ABB RAPID module: Module1.mod

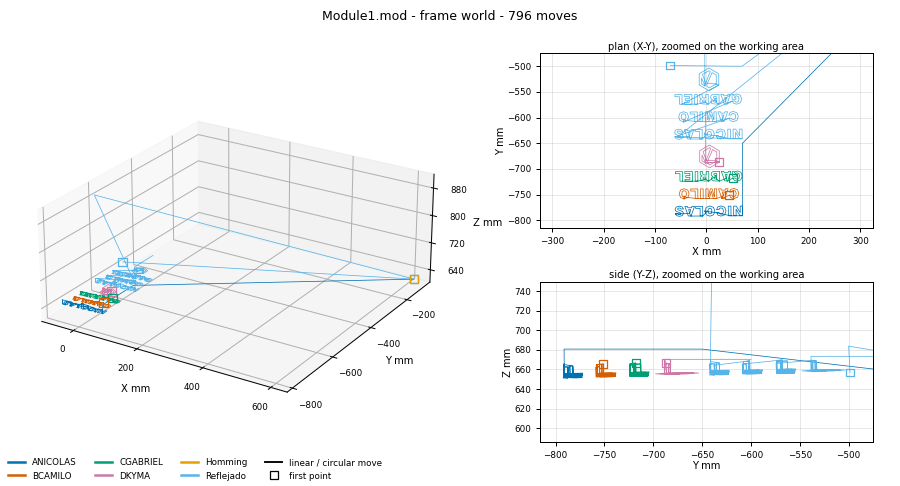
[picture p0: tool path of Module1.mod in frame world, 796 of 800 moves have a stored position in this frame; points joined in program order, loops and branches not executed]
MODULE Module1
    !CONST robtarget Target_10:=[[138.975,143.37,-10],[0.119542298,0.027125582,0.159127158,0.979618492],[-1,-1,1,0],[9E+09,9E+09,9E+09,9E+09,9E+09,9E+09]];
    CONST robtarget Target_10:=[[139.514118203,143.062380794,-24.987379073],[0.119542298,0.027125582,0.159127158,0.979618492],[-1,-1,1,0],[9E+09,9E+09,9E+09,9E+09,9E+09,9E+09]];
    CONST robtarget Target_20:=[[138.975,143.37,0],[0.119542298,0.027125582,0.159127158,0.979618492],[-1,-1,1,0],[9E+09,9E+09,9E+09,9E+09,9E+09,9E+09]];
    CONST robtarget Target_30:=[[133.906,143.37,0],[0.119542298,0.027125582,0.159127158,0.979618492],[-1,-1,1,0],[9E+09,9E+09,9E+09,9E+09,9E+09,9E+09]];
    CONST robtarget Target_40:=[[126.245,130.656,0],[0.119542298,0.027125582,0.159127158,0.979618492],[-1,-1,1,0],[9E+09,9E+09,9E+09,9E+09,9E+09,9E+09]];
    CONST robtarget Target_50:=[[126.245,143.37,0],[0.119542298,0.027125582,0.159127158,0.979618492],[-1,-1,1,0],[9E+09,9E+09,9E+09,9E+09,9E+09,9E+09]];
    CONST robtarget Target_60:=[[121.518,143.37,0],[0.119542298,0.027125582,0.159127158,0.979618492],[-1,-1,1,0],[9E+09,9E+09,9E+09,9E+09,9E+09,9E+09]];
    CONST robtarget Target_70:=[[121.518,124.69,0],[0.119542298,0.027125582,0.159127158,0.979618492],[-1,-1,1,0],[9E+09,9E+09,9E+09,9E+09,9E+09,9E+09]];
    CONST robtarget Target_80:=[[126.603,124.69,0],[0.119542298,0.027125582,0.159127158,0.979618492],[-1,-1,1,0],[9E+09,9E+09,9E+09,9E+09,9E+09,9E+09]];
    CONST robtarget Target_90:=[[134.248,137.371,0],[0.119542298,0.027125582,0.159127158,0.979618492],[-1,-1,1,0],[9E+09,9E+09,9E+09,9E+09,9E+09,9E+09]];
    CONST robtarget Target_100:=[[134.248,124.69,0],[0.119542298,0.027125582,0.159127158,0.979618492],[-1,-1,1,0],[9E+09,9E+09,9E+09,9E+09,9E+09,9E+09]];
    CONST robtarget Target_110:=[[138.975,124.69,0],[0.119542298,0.027125582,0.159127158,0.979618492],[-1,-1,1,0],[9E+09,9E+09,9E+09,9E+09,9E+09,9E+09]];
    CONST robtarget Target_120:=[[138.975,143.37,0],[0.119542298,0.027125582,0.159127158,0.979618492],[-1,-1,1,0],[9E+09,9E+09,9E+09,9E+09,9E+09,9E+09]];
    CONST robtarget Target_130:=[[138.975,143.37,-10],[0.119542298,0.027125582,0.159127158,0.979618492],[-1,-1,1,0],[9E+09,9E+09,9E+09,9E+09,9E+09,9E+09]];
    CONST robtarget Target_140:=[[116.236,143.37,-10],[0.119542298,0.027125582,0.159127158,0.979618492],[-1,-1,1,0],[9E+09,9E+09,9E+09,9E+09,9E+09,9E+09]];
    CONST robtarget Target_150:=[[116.236,143.37,0],[0.119542298,0.027125582,0.159127158,0.979618492],[-1,-1,1,0],[9E+09,9E+09,9E+09,9E+09,9E+09,9E+09]];
    CONST robtarget Target_160:=[[111.069,143.37,0],[0.119542298,0.027125582,0.159127158,0.979618492],[-1,-1,1,0],[9E+09,9E+09,9E+09,9E+09,9E+09,9E+09]];
    CONST robtarget Target_170:=[[111.069,124.69,0],[0.119542298,0.027125582,0.159127158,0.979618492],[-1,-1,1,0],[9E+09,9E+09,9E+09,9E+09,9E+09,9E+09]];
    CONST robtarget Target_180:=[[116.236,124.69,0],[0.119542298,0.027125582,0.159127158,0.979618492],[-1,-1,1,0],[9E+09,9E+09,9E+09,9E+09,9E+09,9E+09]];
    CONST robtarget Target_190:=[[116.236,143.37,0],[0.119542298,0.027125582,0.159127158,0.979618492],[-1,-1,1,0],[9E+09,9E+09,9E+09,9E+09,9E+09,9E+09]];
    CONST robtarget Target_200:=[[116.236,143.37,-10],[0.119542298,0.027125582,0.159127158,0.979618492],[-1,-1,1,0],[9E+09,9E+09,9E+09,9E+09,9E+09,9E+09]];
    CONST robtarget Target_210:=[[88.445,137.143,-10],[0.119542298,0.027125582,0.159127158,0.979618492],[-1,-1,1,0],[9E+09,9E+09,9E+09,9E+09,9E+09,9E+09]];
    CONST robtarget Target_220:=[[88.445,137.143,0],[0.119542298,0.027125582,0.159127158,0.979618492],[-1,-1,1,0],[9E+09,9E+09,9E+09,9E+09,9E+09,9E+09]];
    CONST robtarget Target_230:=[[90.98,142.156,0],[0.119542298,0.027125582,0.159127158,0.979618492],[-1,-1,1,0],[9E+09,9E+09,9E+09,9E+09,9E+09,9E+09]];
    CONST robtarget Target_240:=[[96.97,143.973,0],[0.119542298,0.027125582,0.159127158,0.979618492],[-1,-1,1,0],[9E+09,9E+09,9E+09,9E+09,9E+09,9E+09]];
    CONST robtarget Target_250:=[[104.06,141.341,0],[0.119542298,0.027125582,0.159127158,0.979618492],[-1,-1,1,0],[9E+09,9E+09,9E+09,9E+09,9E+09,9E+09]];
    CONST robtarget Target_260:=[[106.62,134.046,0],[0.119542298,0.027125582,0.159127158,0.979618492],[-1,-1,1,0],[9E+09,9E+09,9E+09,9E+09,9E+09,9E+09]];
    CONST robtarget Target_270:=[[104.077,126.752,0],[0.119542298,0.027125582,0.159127158,0.979618492],[-1,-1,1,0],[9E+09,9E+09,9E+09,9E+09,9E+09,9E+09]];
    CONST robtarget Target_280:=[[96.954,124.136,0],[0.119542298,0.027125582,0.159127158,0.979618492],[-1,-1,1,0],[9E+09,9E+09,9E+09,9E+09,9E+09,9E+09]];
    CONST robtarget Target_290:=[[90.866,125.978,0],[0.119542298,0.027125582,0.159127158,0.979618492],[-1,-1,1,0],[9E+09,9E+09,9E+09,9E+09,9E+09,9E+09]];
    CONST robtarget Target_300:=[[88.201,131.178,0],[0.119542298,0.027125582,0.159127158,0.979618492],[-1,-1,1,0],[9E+09,9E+09,9E+09,9E+09,9E+09,9E+09]];
    CONST robtarget Target_310:=[[90.556,131.178,0],[0.119542298,0.027125582,0.159127158,0.979618492],[-1,-1,1,0],[9E+09,9E+09,9E+09,9E+09,9E+09,9E+09]];
    CONST robtarget Target_320:=[[92.911,131.178,0],[0.119542298,0.027125582,0.159127158,0.979618492],[-1,-1,1,0],[9E+09,9E+09,9E+09,9E+09,9E+09,9E+09]];
    CONST robtarget Target_330:=[[94.207,128.781,0],[0.119542298,0.027125582,0.159127158,0.979618492],[-1,-1,1,0],[9E+09,9E+09,9E+09,9E+09,9E+09,9E+09]];
    CONST robtarget Target_340:=[[96.937,127.885,0],[0.119542298,0.027125582,0.159127158,0.979618492],[-1,-1,1,0],[9E+09,9E+09,9E+09,9E+09,9E+09,9E+09]];
    CONST robtarget Target_350:=[[100.385,129.458,0],[0.119542298,0.027125582,0.159127158,0.979618492],[-1,-1,1,0],[9E+09,9E+09,9E+09,9E+09,9E+09,9E+09]];
    CONST robtarget Target_360:=[[101.583,134.03,0],[0.119542298,0.027125582,0.159127158,0.979618492],[-1,-1,1,0],[9E+09,9E+09,9E+09,9E+09,9E+09,9E+09]];
    CONST robtarget Target_370:=[[100.426,138.635,0],[0.119542298,0.027125582,0.159127158,0.979618492],[-1,-1,1,0],[9E+09,9E+09,9E+09,9E+09,9E+09,9E+09]];
    CONST robtarget Target_380:=[[96.937,140.175,0],[0.119542298,0.027125582,0.159127158,0.979618492],[-1,-1,1,0],[9E+09,9E+09,9E+09,9E+09,9E+09,9E+09]];
    CONST robtarget Target_390:=[[94.329,139.376,0],[0.119542298,0.027125582,0.159127158,0.979618492],[-1,-1,1,0],[9E+09,9E+09,9E+09,9E+09,9E+09,9E+09]];
    CONST robtarget Target_400:=[[93.058,137.143,0],[0.119542298,0.027125582,0.159127158,0.979618492],[-1,-1,1,0],[9E+09,9E+09,9E+09,9E+09,9E+09,9E+09]];
    CONST robtarget Target_410:=[[90.752,137.143,0],[0.119542298,0.027125582,0.159127158,0.979618492],[-1,-1,1,0],[9E+09,9E+09,9E+09,9E+09,9E+09,9E+09]];
    CONST robtarget Target_420:=[[88.445,137.143,0],[0.119542298,0.027125582,0.159127158,0.979618492],[-1,-1,1,0],[9E+09,9E+09,9E+09,9E+09,9E+09,9E+09]];
    CONST robtarget Target_430:=[[88.445,137.143,-10],[0.119542298,0.027125582,0.159127158,0.979618492],[-1,-1,1,0],[9E+09,9E+09,9E+09,9E+09,9E+09,9E+09]];
    CONST robtarget Target_440:=[[65.511,134.046,-10],[0.119542298,0.027125582,0.159127158,0.979618492],[-1,-1,1,0],[9E+09,9E+09,9E+09,9E+09,9E+09,9E+09]];
    CONST robtarget Target_450:=[[65.511,134.046,0],[0.119542298,0.027125582,0.159127158,0.979618492],[-1,-1,1,0],[9E+09,9E+09,9E+09,9E+09,9E+09,9E+09]];
    CONST robtarget Target_460:=[[68.127,141.3,0],[0.119542298,0.027125582,0.159127158,0.979618492],[-1,-1,1,0],[9E+09,9E+09,9E+09,9E+09,9E+09,9E+09]];
    CONST robtarget Target_470:=[[75.21,143.973,0],[0.119542298,0.027125582,0.159127158,0.979618492],[-1,-1,1,0],[9E+09,9E+09,9E+09,9E+09,9E+09,9E+09]];
    CONST robtarget Target_480:=[[82.3,141.3,0],[0.119542298,0.027125582,0.159127158,0.979618492],[-1,-1,1,0],[9E+09,9E+09,9E+09,9E+09,9E+09,9E+09]];
    CONST robtarget Target_490:=[[84.908,134.046,0],[0.119542298,0.027125582,0.159127158,0.979618492],[-1,-1,1,0],[9E+09,9E+09,9E+09,9E+09,9E+09,9E+09]];
    CONST robtarget Target_500:=[[82.3,126.809,0],[0.119542298,0.027125582,0.159127158,0.979618492],[-1,-1,1,0],[9E+09,9E+09,9E+09,9E+09,9E+09,9E+09]];
    CONST robtarget Target_510:=[[75.21,124.136,0],[0.119542298,0.027125582,0.159127158,0.979618492],[-1,-1,1,0],[9E+09,9E+09,9E+09,9E+09,9E+09,9E+09]];
    CONST robtarget Target_520:=[[68.119,126.809,0],[0.119542298,0.027125582,0.159127158,0.979618492],[-1,-1,1,0],[9E+09,9E+09,9E+09,9E+09,9E+09,9E+09]];
    CONST robtarget Target_530:=[[65.511,134.046,0],[0.119542298,0.027125582,0.159127158,0.979618492],[-1,-1,1,0],[9E+09,9E+09,9E+09,9E+09,9E+09,9E+09]];
    CONST robtarget Target_540:=[[65.511,134.046,-10],[0.119542298,0.027125582,0.159127158,0.979618492],[-1,-1,1,0],[9E+09,9E+09,9E+09,9E+09,9E+09,9E+09]];
    CONST robtarget Target_550:=[[71.298,134.046,-10],[0.119542298,0.027125582,0.159127158,0.979618492],[-1,-1,1,0],[9E+09,9E+09,9E+09,9E+09,9E+09,9E+09]];
    CONST robtarget Target_560:=[[71.298,134.046,0],[0.119542298,0.027125582,0.159127158,0.979618492],[-1,-1,1,0],[9E+09,9E+09,9E+09,9E+09,9E+09,9E+09]];
    CONST robtarget Target_570:=[[72.235,129.865,0],[0.119542298,0.027125582,0.159127158,0.979618492],[-1,-1,1,0],[9E+09,9E+09,9E+09,9E+09,9E+09,9E+09]];
    CONST robtarget Target_580:=[[75.193,128.537,0],[0.119542298,0.027125582,0.159127158,0.979618492],[-1,-1,1,0],[9E+09,9E+09,9E+09,9E+09,9E+09,9E+09]];
    CONST robtarget Target_590:=[[78.176,129.865,0],[0.119542298,0.027125582,0.159127158,0.979618492],[-1,-1,1,0],[9E+09,9E+09,9E+09,9E+09,9E+09,9E+09]];
    CONST robtarget Target_600:=[[79.122,134.046,0],[0.119542298,0.027125582,0.159127158,0.979618492],[-1,-1,1,0],[9E+09,9E+09,9E+09,9E+09,9E+09,9E+09]];
    CONST robtarget Target_610:=[[78.176,138.227,0],[0.119542298,0.027125582,0.159127158,0.979618492],[-1,-1,1,0],[9E+09,9E+09,9E+09,9E+09,9E+09,9E+09]];
    CONST robtarget Target_620:=[[75.193,139.556,0],[0.119542298,0.027125582,0.159127158,0.979618492],[-1,-1,1,0],[9E+09,9E+09,9E+09,9E+09,9E+09,9E+09]];
    CONST robtarget Target_630:=[[72.235,138.227,0],[0.119542298,0.027125582,0.159127158,0.979618492],[-1,-1,1,0],[9E+09,9E+09,9E+09,9E+09,9E+09,9E+09]];
    CONST robtarget Target_640:=[[71.298,134.046,0],[0.119542298,0.027125582,0.159127158,0.979618492],[-1,-1,1,0],[9E+09,9E+09,9E+09,9E+09,9E+09,9E+09]];
    CONST robtarget Target_650:=[[71.298,134.046,-10],[0.119542298,0.027125582,0.159127158,0.979618492],[-1,-1,1,0],[9E+09,9E+09,9E+09,9E+09,9E+09,9E+09]];
    CONST robtarget Target_660:=[[61.192,143.37,-10],[0.119542298,0.027125582,0.159127158,0.979618492],[-1,-1,1,0],[9E+09,9E+09,9E+09,9E+09,9E+09,9E+09]];
    CONST robtarget Target_670:=[[61.192,143.37,0],[0.119542298,0.027125582,0.159127158,0.979618492],[-1,-1,1,0],[9E+09,9E+09,9E+09,9E+09,9E+09,9E+09]];
    CONST robtarget Target_680:=[[56.139,143.37,0],[0.119542298,0.027125582,0.159127158,0.979618492],[-1,-1,1,0],[9E+09,9E+09,9E+09,9E+09,9E+09,9E+09]];
    CONST robtarget Target_690:=[[56.139,128.7,0],[0.119542298,0.027125582,0.159127158,0.979618492],[-1,-1,1,0],[9E+09,9E+09,9E+09,9E+09,9E+09,9E+09]];
    CONST robtarget Target_700:=[[47.402,128.7,0],[0.119542298,0.027125582,0.159127158,0.979618492],[-1,-1,1,0],[9E+09,9E+09,9E+09,9E+09,9E+09,9E+09]];
    CONST robtarget Target_710:=[[47.402,124.69,0],[0.119542298,0.027125582,0.159127158,0.979618492],[-1,-1,1,0],[9E+09,9E+09,9E+09,9E+09,9E+09,9E+09]];
    CONST robtarget Target_720:=[[61.192,124.69,0],[0.119542298,0.027125582,0.159127158,0.979618492],[-1,-1,1,0],[9E+09,9E+09,9E+09,9E+09,9E+09,9E+09]];
    CONST robtarget Target_730:=[[61.192,143.37,0],[0.119542298,0.027125582,0.159127158,0.979618492],[-1,-1,1,0],[9E+09,9E+09,9E+09,9E+09,9E+09,9E+09]];
    CONST robtarget Target_740:=[[61.192,143.37,-10],[0.119542298,0.027125582,0.159127158,0.979618492],[-1,-1,1,0],[9E+09,9E+09,9E+09,9E+09,9E+09,9E+09]];
    CONST robtarget Target_750:=[[38.567,143.37,-10],[0.119542298,0.027125582,0.159127158,0.979618492],[-1,-1,1,0],[9E+09,9E+09,9E+09,9E+09,9E+09,9E+09]];
    CONST robtarget Target_760:=[[38.567,143.37,0],[0.119542298,0.027125582,0.159127158,0.979618492],[-1,-1,1,0],[9E+09,9E+09,9E+09,9E+09,9E+09,9E+09]];
    CONST robtarget Target_770:=[[33.025,143.37,0],[0.119542298,0.027125582,0.159127158,0.979618492],[-1,-1,1,0],[9E+09,9E+09,9E+09,9E+09,9E+09,9E+09]];
    CONST robtarget Target_780:=[[26.424,124.69,0],[0.119542298,0.027125582,0.159127158,0.979618492],[-1,-1,1,0],[9E+09,9E+09,9E+09,9E+09,9E+09,9E+09]];
    CONST robtarget Target_790:=[[31.412,124.69,0],[0.119542298,0.027125582,0.159127158,0.979618492],[-1,-1,1,0],[9E+09,9E+09,9E+09,9E+09,9E+09,9E+09]];
    CONST robtarget Target_800:=[[32.178,127.331,0],[0.119542298,0.027125582,0.159127158,0.979618492],[-1,-1,1,0],[9E+09,9E+09,9E+09,9E+09,9E+09,9E+09]];
    CONST robtarget Target_810:=[[39.464,127.331,0],[0.119542298,0.027125582,0.159127158,0.979618492],[-1,-1,1,0],[9E+09,9E+09,9E+09,9E+09,9E+09,9E+09]];
    CONST robtarget Target_820:=[[40.181,124.69,0],[0.119542298,0.027125582,0.159127158,0.979618492],[-1,-1,1,0],[9E+09,9E+09,9E+09,9E+09,9E+09,9E+09]];
    CONST robtarget Target_830:=[[45.169,124.69,0],[0.119542298,0.027125582,0.159127158,0.979618492],[-1,-1,1,0],[9E+09,9E+09,9E+09,9E+09,9E+09,9E+09]];
    CONST robtarget Target_840:=[[38.567,143.37,0],[0.119542298,0.027125582,0.159127158,0.979618492],[-1,-1,1,0],[9E+09,9E+09,9E+09,9E+09,9E+09,9E+09]];
    CONST robtarget Target_850:=[[38.567,143.37,-10],[0.119542298,0.027125582,0.159127158,0.979618492],[-1,-1,1,0],[9E+09,9E+09,9E+09,9E+09,9E+09,9E+09]];
    CONST robtarget Target_860:=[[35.796,138.464,-10],[0.119542298,0.027125582,0.159127158,0.979618492],[-1,-1,1,0],[9E+09,9E+09,9E+09,9E+09,9E+09,9E+09]];
    CONST robtarget Target_870:=[[35.796,138.464,0],[0.119542298,0.027125582,0.159127158,0.979618492],[-1,-1,1,0],[9E+09,9E+09,9E+09,9E+09,9E+09,9E+09]];
    CONST robtarget Target_880:=[[37.834,130.884,0],[0.119542298,0.027125582,0.159127158,0.979618492],[-1,-1,1,0],[9E+09,9E+09,9E+09,9E+09,9E+09,9E+09]];
    CONST robtarget Target_890:=[[33.791,130.884,0],[0.119542298,0.027125582,0.159127158,0.979618492],[-1,-1,1,0],[9E+09,9E+09,9E+09,9E+09,9E+09,9E+09]];
    CONST robtarget Target_900:=[[35.796,138.464,0],[0.119542298,0.027125582,0.159127158,0.979618492],[-1,-1,1,0],[9E+09,9E+09,9E+09,9E+09,9E+09,9E+09]];
    CONST robtarget Target_910:=[[35.796,138.464,-10],[0.119542298,0.027125582,0.159127158,0.979618492],[-1,-1,1,0],[9E+09,9E+09,9E+09,9E+09,9E+09,9E+09]];
    CONST robtarget Target_920:=[[8.038,138.936,-10],[0.119542298,0.027125582,0.159127158,0.979618492],[-1,-1,1,0],[9E+09,9E+09,9E+09,9E+09,9E+09,9E+09]];
    CONST robtarget Target_930:=[[8.038,138.936,0],[0.119542298,0.027125582,0.159127158,0.979618492],[-1,-1,1,0],[9E+09,9E+09,9E+09,9E+09,9E+09,9E+09]];
    CONST robtarget Target_940:=[[10.58,142.702,0],[0.119542298,0.027125582,0.159127158,0.979618492],[-1,-1,1,0],[9E+09,9E+09,9E+09,9E+09,9E+09,9E+09]];
    CONST robtarget Target_950:=[[16.057,143.973,0],[0.119542298,0.027125582,0.159127158,0.979618492],[-1,-1,1,0],[9E+09,9E+09,9E+09,9E+09,9E+09,9E+09]];
    CONST robtarget Target_960:=[[21.558,142.416,0],[0.119542298,0.027125582,0.159127158,0.979618492],[-1,-1,1,0],[9E+09,9E+09,9E+09,9E+09,9E+09,9E+09]];
    CONST robtarget Target_970:=[[23.588,138.219,0],[0.119542298,0.027125582,0.159127158,0.979618492],[-1,-1,1,0],[9E+09,9E+09,9E+09,9E+09,9E+09,9E+09]];
    CONST robtarget Target_980:=[[22.267,134.812,0],[0.119542298,0.027125582,0.159127158,0.979618492],[-1,-1,1,0],[9E+09,9E+09,9E+09,9E+09,9E+09,9E+09]];
    CONST robtarget Target_990:=[[16.611,132.4,0],[0.119542298,0.027125582,0.159127158,0.979618492],[-1,-1,1,0],[9E+09,9E+09,9E+09,9E+09,9E+09,9E+09]];
    CONST robtarget Target_1000:=[[13.16,131.12,0],[0.119542298,0.027125582,0.159127158,0.979618492],[-1,-1,1,0],[9E+09,9E+09,9E+09,9E+09,9E+09,9E+09]];
    CONST robtarget Target_1010:=[[12.324,129.743,0],[0.119542298,0.027125582,0.159127158,0.979618492],[-1,-1,1,0],[9E+09,9E+09,9E+09,9E+09,9E+09,9E+09]];
    CONST robtarget Target_1020:=[[13.172,128.17,0],[0.119542298,0.027125582,0.159127158,0.979618492],[-1,-1,1,0],[9E+09,9E+09,9E+09,9E+09,9E+09,9E+09]];
    CONST robtarget Target_1030:=[[15.633,127.624,0],[0.119542298,0.027125582,0.159127158,0.979618492],[-1,-1,1,0],[9E+09,9E+09,9E+09,9E+09,9E+09,9E+09]];
    CONST robtarget Target_1040:=[[17.858,128.129,0],[0.119542298,0.027125582,0.159127158,0.979618492],[-1,-1,1,0],[9E+09,9E+09,9E+09,9E+09,9E+09,9E+09]];
    CONST robtarget Target_1050:=[[18.926,129.629,0],[0.119542298,0.027125582,0.159127158,0.979618492],[-1,-1,1,0],[9E+09,9E+09,9E+09,9E+09,9E+09,9E+09]];
    CONST robtarget Target_1060:=[[23.783,129.629,0],[0.119542298,0.027125582,0.159127158,0.979618492],[-1,-1,1,0],[9E+09,9E+09,9E+09,9E+09,9E+09,9E+09]];
    CONST robtarget Target_1070:=[[21.192,125.587,0],[0.119542298,0.027125582,0.159127158,0.979618492],[-1,-1,1,0],[9E+09,9E+09,9E+09,9E+09,9E+09,9E+09]];
    CONST robtarget Target_1080:=[[15.715,124.169,0],[0.119542298,0.027125582,0.159127158,0.979618492],[-1,-1,1,0],[9E+09,9E+09,9E+09,9E+09,9E+09,9E+09]];
    CONST robtarget Target_1090:=[[9.554,125.741,0],[0.119542298,0.027125582,0.159127158,0.979618492],[-1,-1,1,0],[9E+09,9E+09,9E+09,9E+09,9E+09,9E+09]];
    CONST robtarget Target_1100:=[[7.451,130.379,0],[0.119542298,0.027125582,0.159127158,0.979618492],[-1,-1,1,0],[9E+09,9E+09,9E+09,9E+09,9E+09,9E+09]];
    CONST robtarget Target_1110:=[[8.885,133.875,0],[0.119542298,0.027125582,0.159127158,0.979618492],[-1,-1,1,0],[9E+09,9E+09,9E+09,9E+09,9E+09,9E+09]];
    CONST robtarget Target_1120:=[[15.03,136.328,0],[0.119542298,0.027125582,0.159127158,0.979618492],[-1,-1,1,0],[9E+09,9E+09,9E+09,9E+09,9E+09,9E+09]];
    CONST robtarget Target_1130:=[[17.85,137.412,0],[0.119542298,0.027125582,0.159127158,0.979618492],[-1,-1,1,0],[9E+09,9E+09,9E+09,9E+09,9E+09,9E+09]];
    CONST robtarget Target_1140:=[[18.698,138.773,0],[0.119542298,0.027125582,0.159127158,0.979618492],[-1,-1,1,0],[9E+09,9E+09,9E+09,9E+09,9E+09,9E+09]];
    CONST robtarget Target_1150:=[[17.972,140.208,0],[0.119542298,0.027125582,0.159127158,0.979618492],[-1,-1,1,0],[9E+09,9E+09,9E+09,9E+09,9E+09,9E+09]];
    CONST robtarget Target_1160:=[[15.976,140.729,0],[0.119542298,0.027125582,0.159127158,0.979618492],[-1,-1,1,0],[9E+09,9E+09,9E+09,9E+09,9E+09,9E+09]];
    CONST robtarget Target_1170:=[[13.889,140.265,0],[0.119542298,0.027125582,0.159127158,0.979618492],[-1,-1,1,0],[9E+09,9E+09,9E+09,9E+09,9E+09,9E+09]];
    CONST robtarget Target_1180:=[[12.879,138.936,0],[0.119542298,0.027125582,0.159127158,0.979618492],[-1,-1,1,0],[9E+09,9E+09,9E+09,9E+09,9E+09,9E+09]];
    CONST robtarget Target_1190:=[[8.038,138.936,0],[0.119542298,0.027125582,0.159127158,0.979618492],[-1,-1,1,0],[9E+09,9E+09,9E+09,9E+09,9E+09,9E+09]];
    CONST robtarget Target_1200:=[[8.038,138.936,-10],[0.119542298,0.027125582,0.159127158,0.979618492],[-1,-1,1,0],[9E+09,9E+09,9E+09,9E+09,9E+09,9E+09]];
    CONST robtarget Target_1210:=[[113.571,103.208,-10],[0.119542298,0.027125582,0.159127158,0.979618492],[-1,-1,1,0],[9E+09,9E+09,9E+09,9E+09,9E+09,9E+09]];
    CONST robtarget Target_1220:=[[113.571,103.208,0],[0.119542298,0.027125582,0.159127158,0.979618492],[-1,-1,1,0],[9E+09,9E+09,9E+09,9E+09,9E+09,9E+09]];
    CONST robtarget Target_1230:=[[116.106,108.22,0],[0.119542298,0.027125582,0.159127158,0.979618492],[-1,-1,1,0],[9E+09,9E+09,9E+09,9E+09,9E+09,9E+09]];
    CONST robtarget Target_1240:=[[122.096,110.037,0],[0.119542298,0.027125582,0.159127158,0.979618492],[-1,-1,1,0],[9E+09,9E+09,9E+09,9E+09,9E+09,9E+09]];
    CONST robtarget Target_1250:=[[129.187,107.405,0],[0.119542298,0.027125582,0.159127158,0.979618492],[-1,-1,1,0],[9E+09,9E+09,9E+09,9E+09,9E+09,9E+09]];
    CONST robtarget Target_1260:=[[131.746,100.111,0],[0.119542298,0.027125582,0.159127158,0.979618492],[-1,-1,1,0],[9E+09,9E+09,9E+09,9E+09,9E+09,9E+09]];
    CONST robtarget Target_1270:=[[129.203,92.817,0],[0.119542298,0.027125582,0.159127158,0.979618492],[-1,-1,1,0],[9E+09,9E+09,9E+09,9E+09,9E+09,9E+09]];
    CONST robtarget Target_1280:=[[122.08,90.2,0],[0.119542298,0.027125582,0.159127158,0.979618492],[-1,-1,1,0],[9E+09,9E+09,9E+09,9E+09,9E+09,9E+09]];
    CONST robtarget Target_1290:=[[115.992,92.042,0],[0.119542298,0.027125582,0.159127158,0.979618492],[-1,-1,1,0],[9E+09,9E+09,9E+09,9E+09,9E+09,9E+09]];
    CONST robtarget Target_1300:=[[113.327,97.242,0],[0.119542298,0.027125582,0.159127158,0.979618492],[-1,-1,1,0],[9E+09,9E+09,9E+09,9E+09,9E+09,9E+09]];
    CONST robtarget Target_1310:=[[118.038,97.242,0],[0.119542298,0.027125582,0.159127158,0.979618492],[-1,-1,1,0],[9E+09,9E+09,9E+09,9E+09,9E+09,9E+09]];
    CONST robtarget Target_1320:=[[119.333,94.846,0],[0.119542298,0.027125582,0.159127158,0.979618492],[-1,-1,1,0],[9E+09,9E+09,9E+09,9E+09,9E+09,9E+09]];
    CONST robtarget Target_1330:=[[122.064,93.949,0],[0.119542298,0.027125582,0.159127158,0.979618492],[-1,-1,1,0],[9E+09,9E+09,9E+09,9E+09,9E+09,9E+09]];
    CONST robtarget Target_1340:=[[125.511,95.522,0],[0.119542298,0.027125582,0.159127158,0.979618492],[-1,-1,1,0],[9E+09,9E+09,9E+09,9E+09,9E+09,9E+09]];
    CONST robtarget Target_1350:=[[126.709,100.094,0],[0.119542298,0.027125582,0.159127158,0.979618492],[-1,-1,1,0],[9E+09,9E+09,9E+09,9E+09,9E+09,9E+09]];
    CONST robtarget Target_1360:=[[125.552,104.699,0],[0.119542298,0.027125582,0.159127158,0.979618492],[-1,-1,1,0],[9E+09,9E+09,9E+09,9E+09,9E+09,9E+09]];
    CONST robtarget Target_1370:=[[122.064,106.239,0],[0.119542298,0.027125582,0.159127158,0.979618492],[-1,-1,1,0],[9E+09,9E+09,9E+09,9E+09,9E+09,9E+09]];
    CONST robtarget Target_1380:=[[119.456,105.441,0],[0.119542298,0.027125582,0.159127158,0.979618492],[-1,-1,1,0],[9E+09,9E+09,9E+09,9E+09,9E+09,9E+09]];
    CONST robtarget Target_1390:=[[118.184,103.208,0],[0.119542298,0.027125582,0.159127158,0.979618492],[-1,-1,1,0],[9E+09,9E+09,9E+09,9E+09,9E+09,9E+09]];
    CONST robtarget Target_1400:=[[113.571,103.208,0],[0.119542298,0.027125582,0.159127158,0.979618492],[-1,-1,1,0],[9E+09,9E+09,9E+09,9E+09,9E+09,9E+09]];
    CONST robtarget Target_1410:=[[113.571,103.208,-10],[0.119542298,0.027125582,0.159127158,0.979618492],[-1,-1,1,0],[9E+09,9E+09,9E+09,9E+09,9E+09,9E+09]];
    CONST robtarget Target_1420:=[[98.771,109.434,-10],[0.119542298,0.027125582,0.159127158,0.979618492],[-1,-1,1,0],[9E+09,9E+09,9E+09,9E+09,9E+09,9E+09]];
    CONST robtarget Target_1430:=[[98.771,109.434,0],[0.119542298,0.027125582,0.159127158,0.979618492],[-1,-1,1,0],[9E+09,9E+09,9E+09,9E+09,9E+09,9E+09]];
    CONST robtarget Target_1440:=[[92.17,90.755,0],[0.119542298,0.027125582,0.159127158,0.979618492],[-1,-1,1,0],[9E+09,9E+09,9E+09,9E+09,9E+09,9E+09]];
    CONST robtarget Target_1450:=[[97.157,90.755,0],[0.119542298,0.027125582,0.159127158,0.979618492],[-1,-1,1,0],[9E+09,9E+09,9E+09,9E+09,9E+09,9E+09]];
    CONST robtarget Target_1460:=[[97.924,93.395,0],[0.119542298,0.027125582,0.159127158,0.979618492],[-1,-1,1,0],[9E+09,9E+09,9E+09,9E+09,9E+09,9E+09]];
    CONST robtarget Target_1470:=[[105.21,93.395,0],[0.119542298,0.027125582,0.159127158,0.979618492],[-1,-1,1,0],[9E+09,9E+09,9E+09,9E+09,9E+09,9E+09]];
    CONST robtarget Target_1480:=[[105.927,90.755,0],[0.119542298,0.027125582,0.159127158,0.979618492],[-1,-1,1,0],[9E+09,9E+09,9E+09,9E+09,9E+09,9E+09]];
    CONST robtarget Target_1490:=[[110.915,90.755,0],[0.119542298,0.027125582,0.159127158,0.979618492],[-1,-1,1,0],[9E+09,9E+09,9E+09,9E+09,9E+09,9E+09]];
    CONST robtarget Target_1500:=[[104.313,109.434,0],[0.119542298,0.027125582,0.159127158,0.979618492],[-1,-1,1,0],[9E+09,9E+09,9E+09,9E+09,9E+09,9E+09]];
    CONST robtarget Target_1510:=[[98.771,109.434,0],[0.119542298,0.027125582,0.159127158,0.979618492],[-1,-1,1,0],[9E+09,9E+09,9E+09,9E+09,9E+09,9E+09]];
    CONST robtarget Target_1520:=[[98.771,109.434,-10],[0.119542298,0.027125582,0.159127158,0.979618492],[-1,-1,1,0],[9E+09,9E+09,9E+09,9E+09,9E+09,9E+09]];
    CONST robtarget Target_1530:=[[101.542,104.528,-10],[0.119542298,0.027125582,0.159127158,0.979618492],[-1,-1,1,0],[9E+09,9E+09,9E+09,9E+09,9E+09,9E+09]];
    CONST robtarget Target_1540:=[[101.542,104.528,0],[0.119542298,0.027125582,0.159127158,0.979618492],[-1,-1,1,0],[9E+09,9E+09,9E+09,9E+09,9E+09,9E+09]];
    CONST robtarget Target_1550:=[[103.58,96.949,0],[0.119542298,0.027125582,0.159127158,0.979618492],[-1,-1,1,0],[9E+09,9E+09,9E+09,9E+09,9E+09,9E+09]];
    CONST robtarget Target_1560:=[[99.537,96.949,0],[0.119542298,0.027125582,0.159127158,0.979618492],[-1,-1,1,0],[9E+09,9E+09,9E+09,9E+09,9E+09,9E+09]];
    CONST robtarget Target_1570:=[[101.542,104.528,0],[0.119542298,0.027125582,0.159127158,0.979618492],[-1,-1,1,0],[9E+09,9E+09,9E+09,9E+09,9E+09,9E+09]];
    CONST robtarget Target_1580:=[[101.542,104.528,-10],[0.119542298,0.027125582,0.159127158,0.979618492],[-1,-1,1,0],[9E+09,9E+09,9E+09,9E+09,9E+09,9E+09]];
    CONST robtarget Target_1590:=[[88.747,109.434,-10],[0.119542298,0.027125582,0.159127158,0.979618492],[-1,-1,1,0],[9E+09,9E+09,9E+09,9E+09,9E+09,9E+09]];
    CONST robtarget Target_1600:=[[88.747,109.434,0],[0.119542298,0.027125582,0.159127158,0.979618492],[-1,-1,1,0],[9E+09,9E+09,9E+09,9E+09,9E+09,9E+09]];
    CONST robtarget Target_1610:=[[88.747,90.755,0],[0.119542298,0.027125582,0.159127158,0.979618492],[-1,-1,1,0],[9E+09,9E+09,9E+09,9E+09,9E+09,9E+09]];
    CONST robtarget Target_1620:=[[84.297,90.755,0],[0.119542298,0.027125582,0.159127158,0.979618492],[-1,-1,1,0],[9E+09,9E+09,9E+09,9E+09,9E+09,9E+09]];
    CONST robtarget Target_1630:=[[84.297,105.848,0],[0.119542298,0.027125582,0.159127158,0.979618492],[-1,-1,1,0],[9E+09,9E+09,9E+09,9E+09,9E+09,9E+09]];
    CONST robtarget Target_1640:=[[83.743,105.848,0],[0.119542298,0.027125582,0.159127158,0.979618492],[-1,-1,1,0],[9E+09,9E+09,9E+09,9E+09,9E+09,9E+09]];
    CONST robtarget Target_1650:=[[79.88,90.755,0],[0.119542298,0.027125582,0.159127158,0.979618492],[-1,-1,1,0],[9E+09,9E+09,9E+09,9E+09,9E+09,9E+09]];
    CONST robtarget Target_1660:=[[76.424,90.755,0],[0.119542298,0.027125582,0.159127158,0.979618492],[-1,-1,1,0],[9E+09,9E+09,9E+09,9E+09,9E+09,9E+09]];
    CONST robtarget Target_1670:=[[72.626,105.848,0],[0.119542298,0.027125582,0.159127158,0.979618492],[-1,-1,1,0],[9E+09,9E+09,9E+09,9E+09,9E+09,9E+09]];
    CONST robtarget Target_1680:=[[71.941,105.848,0],[0.119542298,0.027125582,0.159127158,0.979618492],[-1,-1,1,0],[9E+09,9E+09,9E+09,9E+09,9E+09,9E+09]];
    CONST robtarget Target_1690:=[[71.941,90.755,0],[0.119542298,0.027125582,0.159127158,0.979618492],[-1,-1,1,0],[9E+09,9E+09,9E+09,9E+09,9E+09,9E+09]];
    CONST robtarget Target_1700:=[[67.557,90.755,0],[0.119542298,0.027125582,0.159127158,0.979618492],[-1,-1,1,0],[9E+09,9E+09,9E+09,9E+09,9E+09,9E+09]];
    CONST robtarget Target_1710:=[[67.557,109.434,0],[0.119542298,0.027125582,0.159127158,0.979618492],[-1,-1,1,0],[9E+09,9E+09,9E+09,9E+09,9E+09,9E+09]];
    CONST robtarget Target_1720:=[[74.175,109.434,0],[0.119542298,0.027125582,0.159127158,0.979618492],[-1,-1,1,0],[9E+09,9E+09,9E+09,9E+09,9E+09,9E+09]];
    CONST robtarget Target_1730:=[[78.152,95.482,0],[0.119542298,0.027125582,0.159127158,0.979618492],[-1,-1,1,0],[9E+09,9E+09,9E+09,9E+09,9E+09,9E+09]];
    CONST robtarget Target_1740:=[[82.113,109.434,0],[0.119542298,0.027125582,0.159127158,0.979618492],[-1,-1,1,0],[9E+09,9E+09,9E+09,9E+09,9E+09,9E+09]];
    CONST robtarget Target_1750:=[[88.747,109.434,0],[0.119542298,0.027125582,0.159127158,0.979618492],[-1,-1,1,0],[9E+09,9E+09,9E+09,9E+09,9E+09,9E+09]];
    CONST robtarget Target_1760:=[[88.747,109.434,-10],[0.119542298,0.027125582,0.159127158,0.979618492],[-1,-1,1,0],[9E+09,9E+09,9E+09,9E+09,9E+09,9E+09]];
    CONST robtarget Target_1770:=[[62.308,109.434,-10],[0.119542298,0.027125582,0.159127158,0.979618492],[-1,-1,1,0],[9E+09,9E+09,9E+09,9E+09,9E+09,9E+09]];
    CONST robtarget Target_1780:=[[62.308,109.434,0],[0.119542298,0.027125582,0.159127158,0.979618492],[-1,-1,1,0],[9E+09,9E+09,9E+09,9E+09,9E+09,9E+09]];
    CONST robtarget Target_1790:=[[62.308,90.755,0],[0.119542298,0.027125582,0.159127158,0.979618492],[-1,-1,1,0],[9E+09,9E+09,9E+09,9E+09,9E+09,9E+09]];
    CONST robtarget Target_1800:=[[57.141,90.755,0],[0.119542298,0.027125582,0.159127158,0.979618492],[-1,-1,1,0],[9E+09,9E+09,9E+09,9E+09,9E+09,9E+09]];
    CONST robtarget Target_1810:=[[57.141,109.434,0],[0.119542298,0.027125582,0.159127158,0.979618492],[-1,-1,1,0],[9E+09,9E+09,9E+09,9E+09,9E+09,9E+09]];
    CONST robtarget Target_1820:=[[62.308,109.434,0],[0.119542298,0.027125582,0.159127158,0.979618492],[-1,-1,1,0],[9E+09,9E+09,9E+09,9E+09,9E+09,9E+09]];
    CONST robtarget Target_1830:=[[62.308,109.434,-10],[0.119542298,0.027125582,0.159127158,0.979618492],[-1,-1,1,0],[9E+09,9E+09,9E+09,9E+09,9E+09,9E+09]];
    CONST robtarget Target_1840:=[[51.86,109.434,-10],[0.119542298,0.027125582,0.159127158,0.979618492],[-1,-1,1,0],[9E+09,9E+09,9E+09,9E+09,9E+09,9E+09]];
    CONST robtarget Target_1850:=[[51.86,109.434,0],[0.119542298,0.027125582,0.159127158,0.979618492],[-1,-1,1,0],[9E+09,9E+09,9E+09,9E+09,9E+09,9E+09]];
    CONST robtarget Target_1860:=[[51.86,90.755,0],[0.119542298,0.027125582,0.159127158,0.979618492],[-1,-1,1,0],[9E+09,9E+09,9E+09,9E+09,9E+09,9E+09]];
    CONST robtarget Target_1870:=[[38.07,90.755,0],[0.119542298,0.027125582,0.159127158,0.979618492],[-1,-1,1,0],[9E+09,9E+09,9E+09,9E+09,9E+09,9E+09]];
    CONST robtarget Target_1880:=[[38.07,94.764,0],[0.119542298,0.027125582,0.159127158,0.979618492],[-1,-1,1,0],[9E+09,9E+09,9E+09,9E+09,9E+09,9E+09]];
    CONST robtarget Target_1890:=[[46.807,94.764,0],[0.119542298,0.027125582,0.159127158,0.979618492],[-1,-1,1,0],[9E+09,9E+09,9E+09,9E+09,9E+09,9E+09]];
    CONST robtarget Target_1900:=[[46.807,109.434,0],[0.119542298,0.027125582,0.159127158,0.979618492],[-1,-1,1,0],[9E+09,9E+09,9E+09,9E+09,9E+09,9E+09]];
    CONST robtarget Target_1910:=[[51.86,109.434,0],[0.119542298,0.027125582,0.159127158,0.979618492],[-1,-1,1,0],[9E+09,9E+09,9E+09,9E+09,9E+09,9E+09]];
    CONST robtarget Target_1920:=[[51.86,109.434,-10],[0.119542298,0.027125582,0.159127158,0.979618492],[-1,-1,1,0],[9E+09,9E+09,9E+09,9E+09,9E+09,9E+09]];
    CONST robtarget Target_1930:=[[25.242,106.256,-10],[0.119542298,0.027125582,0.159127158,0.979618492],[-1,-1,1,0],[9E+09,9E+09,9E+09,9E+09,9E+09,9E+09]];
    CONST robtarget Target_1940:=[[25.242,106.256,0],[0.119542298,0.027125582,0.159127158,0.979618492],[-1,-1,1,0],[9E+09,9E+09,9E+09,9E+09,9E+09,9E+09]];
    CONST robtarget Target_1950:=[[28.739,104.772,0],[0.119542298,0.027125582,0.159127158,0.979618492],[-1,-1,1,0],[9E+09,9E+09,9E+09,9E+09,9E+09,9E+09]];
    CONST robtarget Target_1960:=[[29.855,100.111,0],[0.119542298,0.027125582,0.159127158,0.979618492],[-1,-1,1,0],[9E+09,9E+09,9E+09,9E+09,9E+09,9E+09]];
    CONST robtarget Target_1970:=[[28.739,95.449,0],[0.119542298,0.027125582,0.159127158,0.979618492],[-1,-1,1,0],[9E+09,9E+09,9E+09,9E+09,9E+09,9E+09]];
    CONST robtarget Target_1980:=[[25.242,93.966,0],[0.119542298,0.027125582,0.159127158,0.979618492],[-1,-1,1,0],[9E+09,9E+09,9E+09,9E+09,9E+09,9E+09]];
    CONST robtarget Target_1990:=[[21.754,95.441,0],[0.119542298,0.027125582,0.159127158,0.979618492],[-1,-1,1,0],[9E+09,9E+09,9E+09,9E+09,9E+09,9E+09]];
    CONST robtarget Target_2000:=[[20.646,100.111,0],[0.119542298,0.027125582,0.159127158,0.979618492],[-1,-1,1,0],[9E+09,9E+09,9E+09,9E+09,9E+09,9E+09]];
    CONST robtarget Target_2010:=[[21.754,104.772,0],[0.119542298,0.027125582,0.159127158,0.979618492],[-1,-1,1,0],[9E+09,9E+09,9E+09,9E+09,9E+09,9E+09]];
    CONST robtarget Target_2020:=[[25.242,106.256,0],[0.119542298,0.027125582,0.159127158,0.979618492],[-1,-1,1,0],[9E+09,9E+09,9E+09,9E+09,9E+09,9E+09]];
    CONST robtarget Target_2030:=[[25.242,106.256,-10],[0.119542298,0.027125582,0.159127158,0.979618492],[-1,-1,1,0],[9E+09,9E+09,9E+09,9E+09,9E+09,9E+09]];
    CONST robtarget Target_2040:=[[25.258,110.037,-10],[0.119542298,0.027125582,0.159127158,0.979618492],[-1,-1,1,0],[9E+09,9E+09,9E+09,9E+09,9E+09,9E+09]];
    CONST robtarget Target_2050:=[[25.258,110.037,0],[0.119542298,0.027125582,0.159127158,0.979618492],[-1,-1,1,0],[9E+09,9E+09,9E+09,9E+09,9E+09,9E+09]];
    CONST robtarget Target_2060:=[[18.176,107.364,0],[0.119542298,0.027125582,0.159127158,0.979618492],[-1,-1,1,0],[9E+09,9E+09,9E+09,9E+09,9E+09,9E+09]];
    CONST robtarget Target_2070:=[[15.56,100.111,0],[0.119542298,0.027125582,0.159127158,0.979618492],[-1,-1,1,0],[9E+09,9E+09,9E+09,9E+09,9E+09,9E+09]];
    CONST robtarget Target_2080:=[[18.168,92.874,0],[0.119542298,0.027125582,0.159127158,0.979618492],[-1,-1,1,0],[9E+09,9E+09,9E+09,9E+09,9E+09,9E+09]];
    CONST robtarget Target_2090:=[[25.258,90.2,0],[0.119542298,0.027125582,0.159127158,0.979618492],[-1,-1,1,0],[9E+09,9E+09,9E+09,9E+09,9E+09,9E+09]];
    CONST robtarget Target_2100:=[[32.349,92.874,0],[0.119542298,0.027125582,0.159127158,0.979618492],[-1,-1,1,0],[9E+09,9E+09,9E+09,9E+09,9E+09,9E+09]];
    CONST robtarget Target_2110:=[[34.957,100.111,0],[0.119542298,0.027125582,0.159127158,0.979618492],[-1,-1,1,0],[9E+09,9E+09,9E+09,9E+09,9E+09,9E+09]];
    CONST robtarget Target_2120:=[[32.349,107.364,0],[0.119542298,0.027125582,0.159127158,0.979618492],[-1,-1,1,0],[9E+09,9E+09,9E+09,9E+09,9E+09,9E+09]];
    CONST robtarget Target_2130:=[[25.258,110.037,0],[0.119542298,0.027125582,0.159127158,0.979618492],[-1,-1,1,0],[9E+09,9E+09,9E+09,9E+09,9E+09,9E+09]];
    CONST robtarget Target_2140:=[[25.258,110.037,-10],[0.119542298,0.027125582,0.159127158,0.979618492],[-1,-1,1,0],[9E+09,9E+09,9E+09,9E+09,9E+09,9E+09]];
    CONST robtarget Target_2150:=[[120.369,69.924,-10],[0.119542298,0.027125582,0.159127158,0.979618492],[-1,-1,1,0],[9E+09,9E+09,9E+09,9E+09,9E+09,9E+09]];
    CONST robtarget Target_2160:=[[120.369,69.924,0],[0.119542298,0.027125582,0.159127158,0.979618492],[-1,-1,1,0],[9E+09,9E+09,9E+09,9E+09,9E+09,9E+09]];
    CONST robtarget Target_2170:=[[125.21,69.924,0],[0.119542298,0.027125582,0.159127158,0.979618492],[-1,-1,1,0],[9E+09,9E+09,9E+09,9E+09,9E+09,9E+09]];
    CONST robtarget Target_2180:=[[126.514,71.717,0],[0.119542298,0.027125582,0.159127158,0.979618492],[-1,-1,1,0],[9E+09,9E+09,9E+09,9E+09,9E+09,9E+09]];
    CONST robtarget Target_2190:=[[128.763,72.337,0],[0.119542298,0.027125582,0.159127158,0.979618492],[-1,-1,1,0],[9E+09,9E+09,9E+09,9E+09,9E+09,9E+09]];
    CONST robtarget Target_2200:=[[132.178,70.715,0],[0.119542298,0.027125582,0.159127158,0.979618492],[-1,-1,1,0],[9E+09,9E+09,9E+09,9E+09,9E+09,9E+09]];
    CONST robtarget Target_2210:=[[133.376,66.061,0],[0.119542298,0.027125582,0.159127158,0.979618492],[-1,-1,1,0],[9E+09,9E+09,9E+09,9E+09,9E+09,9E+09]];
    CONST robtarget Target_2220:=[[132.243,61.367,0],[0.119542298,0.027125582,0.159127158,0.979618492],[-1,-1,1,0],[9E+09,9E+09,9E+09,9E+09,9E+09,9E+09]];
    CONST robtarget Target_2230:=[[128.763,59.834,0],[0.119542298,0.027125582,0.159127158,0.979618492],[-1,-1,1,0],[9E+09,9E+09,9E+09,9E+09,9E+09,9E+09]];
    CONST robtarget Target_2240:=[[125.723,60.861,0],[0.119542298,0.027125582,0.159127158,0.979618492],[-1,-1,1,0],[9E+09,9E+09,9E+09,9E+09,9E+09,9E+09]];
    CONST robtarget Target_2250:=[[124.46,63.486,0],[0.119542298,0.027125582,0.159127158,0.979618492],[-1,-1,1,0],[9E+09,9E+09,9E+09,9E+09,9E+09,9E+09]];
    CONST robtarget Target_2260:=[[125.927,63.494,0],[0.119542298,0.027125582,0.159127158,0.979618492],[-1,-1,1,0],[9E+09,9E+09,9E+09,9E+09,9E+09,9E+09]];
    CONST robtarget Target_2270:=[[127.394,63.502,0],[0.119542298,0.027125582,0.159127158,0.979618492],[-1,-1,1,0],[9E+09,9E+09,9E+09,9E+09,9E+09,9E+09]];
    CONST robtarget Target_2280:=[[127.394,66.501,0],[0.119542298,0.027125582,0.159127158,0.979618492],[-1,-1,1,0],[9E+09,9E+09,9E+09,9E+09,9E+09,9E+09]];
    CONST robtarget Target_2290:=[[119.961,66.501,0],[0.119542298,0.027125582,0.159127158,0.979618492],[-1,-1,1,0],[9E+09,9E+09,9E+09,9E+09,9E+09,9E+09]];
    CONST robtarget Target_2300:=[[119.961,56.819,0],[0.119542298,0.027125582,0.159127158,0.979618492],[-1,-1,1,0],[9E+09,9E+09,9E+09,9E+09,9E+09,9E+09]];
    CONST robtarget Target_2310:=[[122.928,56.819,0],[0.119542298,0.027125582,0.159127158,0.979618492],[-1,-1,1,0],[9E+09,9E+09,9E+09,9E+09,9E+09,9E+09]];
    CONST robtarget Target_2320:=[[123.433,59.557,0],[0.119542298,0.027125582,0.159127158,0.979618492],[-1,-1,1,0],[9E+09,9E+09,9E+09,9E+09,9E+09,9E+09]];
    CONST robtarget Target_2330:=[[125.78,57.129,0],[0.119542298,0.027125582,0.159127158,0.979618492],[-1,-1,1,0],[9E+09,9E+09,9E+09,9E+09,9E+09,9E+09]];
    CONST robtarget Target_2340:=[[129.855,56.265,0],[0.119542298,0.027125582,0.159127158,0.979618492],[-1,-1,1,0],[9E+09,9E+09,9E+09,9E+09,9E+09,9E+09]];
    CONST robtarget Target_2350:=[[136.155,58.938,0],[0.119542298,0.027125582,0.159127158,0.979618492],[-1,-1,1,0],[9E+09,9E+09,9E+09,9E+09,9E+09,9E+09]];
    CONST robtarget Target_2360:=[[138.478,66.175,0],[0.119542298,0.027125582,0.159127158,0.979618492],[-1,-1,1,0],[9E+09,9E+09,9E+09,9E+09,9E+09,9E+09]];
    CONST robtarget Target_2370:=[[135.91,73.469,0],[0.119542298,0.027125582,0.159127158,0.979618492],[-1,-1,1,0],[9E+09,9E+09,9E+09,9E+09,9E+09,9E+09]];
    CONST robtarget Target_2380:=[[128.796,76.102,0],[0.119542298,0.027125582,0.159127158,0.979618492],[-1,-1,1,0],[9E+09,9E+09,9E+09,9E+09,9E+09,9E+09]];
    CONST robtarget Target_2390:=[[123.148,74.48,0],[0.119542298,0.027125582,0.159127158,0.979618492],[-1,-1,1,0],[9E+09,9E+09,9E+09,9E+09,9E+09,9E+09]];
    CONST robtarget Target_2400:=[[120.369,69.924,0],[0.119542298,0.027125582,0.159127158,0.979618492],[-1,-1,1,0],[9E+09,9E+09,9E+09,9E+09,9E+09,9E+09]];
    CONST robtarget Target_2410:=[[120.369,69.924,-10],[0.119542298,0.027125582,0.159127158,0.979618492],[-1,-1,1,0],[9E+09,9E+09,9E+09,9E+09,9E+09,9E+09]];
    CONST robtarget Target_2420:=[[110.1,75.499,-10],[0.119542298,0.027125582,0.159127158,0.979618492],[-1,-1,1,0],[9E+09,9E+09,9E+09,9E+09,9E+09,9E+09]];
    CONST robtarget Target_2430:=[[110.1,75.499,0],[0.119542298,0.027125582,0.159127158,0.979618492],[-1,-1,1,0],[9E+09,9E+09,9E+09,9E+09,9E+09,9E+09]];
    CONST robtarget Target_2440:=[[104.558,75.499,0],[0.119542298,0.027125582,0.159127158,0.979618492],[-1,-1,1,0],[9E+09,9E+09,9E+09,9E+09,9E+09,9E+09]];
    CONST robtarget Target_2450:=[[97.956,56.819,0],[0.119542298,0.027125582,0.159127158,0.979618492],[-1,-1,1,0],[9E+09,9E+09,9E+09,9E+09,9E+09,9E+09]];
    CONST robtarget Target_2460:=[[102.944,56.819,0],[0.119542298,0.027125582,0.159127158,0.979618492],[-1,-1,1,0],[9E+09,9E+09,9E+09,9E+09,9E+09,9E+09]];
    CONST robtarget Target_2470:=[[103.71,59.46,0],[0.119542298,0.027125582,0.159127158,0.979618492],[-1,-1,1,0],[9E+09,9E+09,9E+09,9E+09,9E+09,9E+09]];
    CONST robtarget Target_2480:=[[110.996,59.46,0],[0.119542298,0.027125582,0.159127158,0.979618492],[-1,-1,1,0],[9E+09,9E+09,9E+09,9E+09,9E+09,9E+09]];
    CONST robtarget Target_2490:=[[111.713,56.819,0],[0.119542298,0.027125582,0.159127158,0.979618492],[-1,-1,1,0],[9E+09,9E+09,9E+09,9E+09,9E+09,9E+09]];
    CONST robtarget Target_2500:=[[116.701,56.819,0],[0.119542298,0.027125582,0.159127158,0.979618492],[-1,-1,1,0],[9E+09,9E+09,9E+09,9E+09,9E+09,9E+09]];
    CONST robtarget Target_2510:=[[110.1,75.499,0],[0.119542298,0.027125582,0.159127158,0.979618492],[-1,-1,1,0],[9E+09,9E+09,9E+09,9E+09,9E+09,9E+09]];
    CONST robtarget Target_2520:=[[110.1,75.499,-10],[0.119542298,0.027125582,0.159127158,0.979618492],[-1,-1,1,0],[9E+09,9E+09,9E+09,9E+09,9E+09,9E+09]];
    CONST robtarget Target_2530:=[[107.329,70.592,-10],[0.119542298,0.027125582,0.159127158,0.979618492],[-1,-1,1,0],[9E+09,9E+09,9E+09,9E+09,9E+09,9E+09]];
    CONST robtarget Target_2540:=[[107.329,70.592,0],[0.119542298,0.027125582,0.159127158,0.979618492],[-1,-1,1,0],[9E+09,9E+09,9E+09,9E+09,9E+09,9E+09]];
    CONST robtarget Target_2550:=[[109.366,63.013,0],[0.119542298,0.027125582,0.159127158,0.979618492],[-1,-1,1,0],[9E+09,9E+09,9E+09,9E+09,9E+09,9E+09]];
    CONST robtarget Target_2560:=[[105.324,63.013,0],[0.119542298,0.027125582,0.159127158,0.979618492],[-1,-1,1,0],[9E+09,9E+09,9E+09,9E+09,9E+09,9E+09]];
    CONST robtarget Target_2570:=[[107.329,70.592,0],[0.119542298,0.027125582,0.159127158,0.979618492],[-1,-1,1,0],[9E+09,9E+09,9E+09,9E+09,9E+09,9E+09]];
    CONST robtarget Target_2580:=[[107.329,70.592,-10],[0.119542298,0.027125582,0.159127158,0.979618492],[-1,-1,1,0],[9E+09,9E+09,9E+09,9E+09,9E+09,9E+09]];
    CONST robtarget Target_2590:=[[94.533,75.499,-10],[0.119542298,0.027125582,0.159127158,0.979618492],[-1,-1,1,0],[9E+09,9E+09,9E+09,9E+09,9E+09,9E+09]];
    CONST robtarget Target_2600:=[[94.533,75.499,0],[0.119542298,0.027125582,0.159127158,0.979618492],[-1,-1,1,0],[9E+09,9E+09,9E+09,9E+09,9E+09,9E+09]];
    CONST robtarget Target_2610:=[[86.921,75.499,0],[0.119542298,0.027125582,0.159127158,0.979618492],[-1,-1,1,0],[9E+09,9E+09,9E+09,9E+09,9E+09,9E+09]];
    CONST robtarget Target_2620:=[[81.379,74.944,0],[0.119542298,0.027125582,0.159127158,0.979618492],[-1,-1,1,0],[9E+09,9E+09,9E+09,9E+09,9E+09,9E+09]];
    CONST robtarget Target_2630:=[[79.366,73.355,0],[0.119542298,0.027125582,0.159127158,0.979618492],[-1,-1,1,0],[9E+09,9E+09,9E+09,9E+09,9E+09,9E+09]];
    CONST robtarget Target_2640:=[[78.624,70.804,0],[0.119542298,0.027125582,0.159127158,0.979618492],[-1,-1,1,0],[9E+09,9E+09,9E+09,9E+09,9E+09,9E+09]];
    CONST robtarget Target_2650:=[[79.382,68.433,0],[0.119542298,0.027125582,0.159127158,0.979618492],[-1,-1,1,0],[9E+09,9E+09,9E+09,9E+09,9E+09,9E+09]];
    CONST robtarget Target_2660:=[[81.509,66.795,0],[0.119542298,0.027125582,0.159127158,0.979618492],[-1,-1,1,0],[9E+09,9E+09,9E+09,9E+09,9E+09,9E+09]];
    CONST robtarget Target_2670:=[[78.869,64.993,0],[0.119542298,0.027125582,0.159127158,0.979618492],[-1,-1,1,0],[9E+09,9E+09,9E+09,9E+09,9E+09,9E+09]];
    CONST robtarget Target_2680:=[[78.005,61.986,0],[0.119542298,0.027125582,0.159127158,0.979618492],[-1,-1,1,0],[9E+09,9E+09,9E+09,9E+09,9E+09,9E+09]];
    CONST robtarget Target_2690:=[[78.673,59.394,0],[0.119542298,0.027125582,0.159127158,0.979618492],[-1,-1,1,0],[9E+09,9E+09,9E+09,9E+09,9E+09,9E+09]];
    CONST robtarget Target_2700:=[[80.564,57.667,0],[0.119542298,0.027125582,0.159127158,0.979618492],[-1,-1,1,0],[9E+09,9E+09,9E+09,9E+09,9E+09,9E+09]];
    CONST robtarget Target_2710:=[[82.577,57.015,0],[0.119542298,0.027125582,0.159127158,0.979618492],[-1,-1,1,0],[9E+09,9E+09,9E+09,9E+09,9E+09,9E+09]];
    CONST robtarget Target_2720:=[[86.122,56.819,0],[0.119542298,0.027125582,0.159127158,0.979618492],[-1,-1,1,0],[9E+09,9E+09,9E+09,9E+09,9E+09,9E+09]];
    CONST robtarget Target_2730:=[[94.533,56.819,0],[0.119542298,0.027125582,0.159127158,0.979618492],[-1,-1,1,0],[9E+09,9E+09,9E+09,9E+09,9E+09,9E+09]];
    CONST robtarget Target_2740:=[[94.533,75.499,0],[0.119542298,0.027125582,0.159127158,0.979618492],[-1,-1,1,0],[9E+09,9E+09,9E+09,9E+09,9E+09,9E+09]];
    CONST robtarget Target_2750:=[[94.533,75.499,-10],[0.119542298,0.027125582,0.159127158,0.979618492],[-1,-1,1,0],[9E+09,9E+09,9E+09,9E+09,9E+09,9E+09]];
    CONST robtarget Target_2760:=[[88.991,71.652,-10],[0.119542298,0.027125582,0.159127158,0.979618492],[-1,-1,1,0],[9E+09,9E+09,9E+09,9E+09,9E+09,9E+09]];
    CONST robtarget Target_2770:=[[88.991,71.652,0],[0.119542298,0.027125582,0.159127158,0.979618492],[-1,-1,1,0],[9E+09,9E+09,9E+09,9E+09,9E+09,9E+09]];
    CONST robtarget Target_2780:=[[87.214,71.652,0],[0.119542298,0.027125582,0.159127158,0.979618492],[-1,-1,1,0],[9E+09,9E+09,9E+09,9E+09,9E+09,9E+09]];
    CONST robtarget Target_2790:=[[84.501,71.285,0],[0.119542298,0.027125582,0.159127158,0.979618492],[-1,-1,1,0],[9E+09,9E+09,9E+09,9E+09,9E+09,9E+09]];
    CONST robtarget Target_2800:=[[83.922,69.924,0],[0.119542298,0.027125582,0.159127158,0.979618492],[-1,-1,1,0],[9E+09,9E+09,9E+09,9E+09,9E+09,9E+09]];
    CONST robtarget Target_2810:=[[84.468,68.596,0],[0.119542298,0.027125582,0.159127158,0.979618492],[-1,-1,1,0],[9E+09,9E+09,9E+09,9E+09,9E+09,9E+09]];
    CONST robtarget Target_2820:=[[86.334,68.196,0],[0.119542298,0.027125582,0.159127158,0.979618492],[-1,-1,1,0],[9E+09,9E+09,9E+09,9E+09,9E+09,9E+09]];
    CONST robtarget Target_2830:=[[87.663,68.196,0],[0.119542298,0.027125582,0.159127158,0.979618492],[-1,-1,1,0],[9E+09,9E+09,9E+09,9E+09,9E+09,9E+09]];
    CONST robtarget Target_2840:=[[88.991,68.196,0],[0.119542298,0.027125582,0.159127158,0.979618492],[-1,-1,1,0],[9E+09,9E+09,9E+09,9E+09,9E+09,9E+09]];
    CONST robtarget Target_2850:=[[88.991,71.652,0],[0.119542298,0.027125582,0.159127158,0.979618492],[-1,-1,1,0],[9E+09,9E+09,9E+09,9E+09,9E+09,9E+09]];
    CONST robtarget Target_2860:=[[88.991,71.652,-10],[0.119542298,0.027125582,0.159127158,0.979618492],[-1,-1,1,0],[9E+09,9E+09,9E+09,9E+09,9E+09,9E+09]];
    CONST robtarget Target_2870:=[[88.991,64.545,-10],[0.119542298,0.027125582,0.159127158,0.979618492],[-1,-1,1,0],[9E+09,9E+09,9E+09,9E+09,9E+09,9E+09]];
    CONST robtarget Target_2880:=[[88.991,64.545,0],[0.119542298,0.027125582,0.159127158,0.979618492],[-1,-1,1,0],[9E+09,9E+09,9E+09,9E+09,9E+09,9E+09]];
    CONST robtarget Target_2890:=[[87.532,64.545,0],[0.119542298,0.027125582,0.159127158,0.979618492],[-1,-1,1,0],[9E+09,9E+09,9E+09,9E+09,9E+09,9E+09]];
    CONST robtarget Target_2900:=[[86.073,64.545,0],[0.119542298,0.027125582,0.159127158,0.979618492],[-1,-1,1,0],[9E+09,9E+09,9E+09,9E+09,9E+09,9E+09]];
    CONST robtarget Target_2910:=[[83.922,64.121,0],[0.119542298,0.027125582,0.159127158,0.979618492],[-1,-1,1,0],[9E+09,9E+09,9E+09,9E+09,9E+09,9E+09]];
    CONST robtarget Target_2920:=[[83.286,62.72,0],[0.119542298,0.027125582,0.159127158,0.979618492],[-1,-1,1,0],[9E+09,9E+09,9E+09,9E+09,9E+09,9E+09]];
    CONST robtarget Target_2930:=[[83.906,61.285,0],[0.119542298,0.027125582,0.159127158,0.979618492],[-1,-1,1,0],[9E+09,9E+09,9E+09,9E+09,9E+09,9E+09]];
    CONST robtarget Target_2940:=[[86.008,60.861,0],[0.119542298,0.027125582,0.159127158,0.979618492],[-1,-1,1,0],[9E+09,9E+09,9E+09,9E+09,9E+09,9E+09]];
    CONST robtarget Target_2950:=[[87.5,60.861,0],[0.119542298,0.027125582,0.159127158,0.979618492],[-1,-1,1,0],[9E+09,9E+09,9E+09,9E+09,9E+09,9E+09]];
    CONST robtarget Target_2960:=[[88.991,60.861,0],[0.119542298,0.027125582,0.159127158,0.979618492],[-1,-1,1,0],[9E+09,9E+09,9E+09,9E+09,9E+09,9E+09]];
    CONST robtarget Target_2970:=[[88.991,64.545,0],[0.119542298,0.027125582,0.159127158,0.979618492],[-1,-1,1,0],[9E+09,9E+09,9E+09,9E+09,9E+09,9E+09]];
    CONST robtarget Target_2980:=[[88.991,64.545,-10],[0.119542298,0.027125582,0.159127158,0.979618492],[-1,-1,1,0],[9E+09,9E+09,9E+09,9E+09,9E+09,9E+09]];
    CONST robtarget Target_2990:=[[73.457,75.499,-10],[0.119542298,0.027125582,0.159127158,0.979618492],[-1,-1,1,0],[9E+09,9E+09,9E+09,9E+09,9E+09,9E+09]];
    CONST robtarget Target_3000:=[[73.457,75.499,0],[0.119542298,0.027125582,0.159127158,0.979618492],[-1,-1,1,0],[9E+09,9E+09,9E+09,9E+09,9E+09,9E+09]];
    CONST robtarget Target_3010:=[[65.258,75.499,0],[0.119542298,0.027125582,0.159127158,0.979618492],[-1,-1,1,0],[9E+09,9E+09,9E+09,9E+09,9E+09,9E+09]];
    CONST robtarget Target_3020:=[[58.665,74.358,0],[0.119542298,0.027125582,0.159127158,0.979618492],[-1,-1,1,0],[9E+09,9E+09,9E+09,9E+09,9E+09,9E+09]];
    CONST robtarget Target_3030:=[[56.913,70.446,0],[0.119542298,0.027125582,0.159127158,0.979618492],[-1,-1,1,0],[9E+09,9E+09,9E+09,9E+09,9E+09,9E+09]];
    CONST robtarget Target_3040:=[[57.785,67.324,0],[0.119542298,0.027125582,0.159127158,0.979618492],[-1,-1,1,0],[9E+09,9E+09,9E+09,9E+09,9E+09,9E+09]];
    CONST robtarget Target_3050:=[[60.613,65.474,0],[0.119542298,0.027125582,0.159127158,0.979618492],[-1,-1,1,0],[9E+09,9E+09,9E+09,9E+09,9E+09,9E+09]];
    CONST robtarget Target_3060:=[[57.736,63.95,0],[0.119542298,0.027125582,0.159127158,0.979618492],[-1,-1,1,0],[9E+09,9E+09,9E+09,9E+09,9E+09,9E+09]];
    CONST robtarget Target_3070:=[[56.88,61.024,0],[0.119542298,0.027125582,0.159127158,0.979618492],[-1,-1,1,0],[9E+09,9E+09,9E+09,9E+09,9E+09,9E+09]];
    CONST robtarget Target_3080:=[[56.799,58.115,0],[0.119542298,0.027125582,0.159127158,0.979618492],[-1,-1,1,0],[9E+09,9E+09,9E+09,9E+09,9E+09,9E+09]];
    CONST robtarget Target_3090:=[[56.424,56.819,0],[0.119542298,0.027125582,0.159127158,0.979618492],[-1,-1,1,0],[9E+09,9E+09,9E+09,9E+09,9E+09,9E+09]];
    CONST robtarget Target_3100:=[[61.395,56.819,0],[0.119542298,0.027125582,0.159127158,0.979618492],[-1,-1,1,0],[9E+09,9E+09,9E+09,9E+09,9E+09,9E+09]];
    CONST robtarget Target_3110:=[[61.656,58.27,0],[0.119542298,0.027125582,0.159127158,0.979618492],[-1,-1,1,0],[9E+09,9E+09,9E+09,9E+09,9E+09,9E+09]];
    CONST robtarget Target_3120:=[[61.656,59.394,0],[0.119542298,0.027125582,0.159127158,0.979618492],[-1,-1,1,0],[9E+09,9E+09,9E+09,9E+09,9E+09,9E+09]];
    CONST robtarget Target_3130:=[[61.656,60.519,0],[0.119542298,0.027125582,0.159127158,0.979618492],[-1,-1,1,0],[9E+09,9E+09,9E+09,9E+09,9E+09,9E+09]];
    CONST robtarget Target_3140:=[[62.43,62.923,0],[0.119542298,0.027125582,0.159127158,0.979618492],[-1,-1,1,0],[9E+09,9E+09,9E+09,9E+09,9E+09,9E+09]];
    CONST robtarget Target_3150:=[[64.737,63.714,0],[0.119542298,0.027125582,0.159127158,0.979618492],[-1,-1,1,0],[9E+09,9E+09,9E+09,9E+09,9E+09,9E+09]];
    CONST robtarget Target_3160:=[[68.486,63.714,0],[0.119542298,0.027125582,0.159127158,0.979618492],[-1,-1,1,0],[9E+09,9E+09,9E+09,9E+09,9E+09,9E+09]];
    CONST robtarget Target_3170:=[[68.486,56.819,0],[0.119542298,0.027125582,0.159127158,0.979618492],[-1,-1,1,0],[9E+09,9E+09,9E+09,9E+09,9E+09,9E+09]];
    CONST robtarget Target_3180:=[[73.457,56.819,0],[0.119542298,0.027125582,0.159127158,0.979618492],[-1,-1,1,0],[9E+09,9E+09,9E+09,9E+09,9E+09,9E+09]];
    CONST robtarget Target_3190:=[[73.457,75.499,0],[0.119542298,0.027125582,0.159127158,0.979618492],[-1,-1,1,0],[9E+09,9E+09,9E+09,9E+09,9E+09,9E+09]];
    CONST robtarget Target_3200:=[[73.457,75.499,-10],[0.119542298,0.027125582,0.159127158,0.979618492],[-1,-1,1,0],[9E+09,9E+09,9E+09,9E+09,9E+09,9E+09]];
    CONST robtarget Target_3210:=[[67.801,71.342,-10],[0.119542298,0.027125582,0.159127158,0.979618492],[-1,-1,1,0],[9E+09,9E+09,9E+09,9E+09,9E+09,9E+09]];
    CONST robtarget Target_3220:=[[67.801,71.342,0],[0.119542298,0.027125582,0.159127158,0.979618492],[-1,-1,1,0],[9E+09,9E+09,9E+09,9E+09,9E+09,9E+09]];
    CONST robtarget Target_3230:=[[65.047,71.342,0],[0.119542298,0.027125582,0.159127158,0.979618492],[-1,-1,1,0],[9E+09,9E+09,9E+09,9E+09,9E+09,9E+09]];
    CONST robtarget Target_3240:=[[62.74,70.918,0],[0.119542298,0.027125582,0.159127158,0.979618492],[-1,-1,1,0],[9E+09,9E+09,9E+09,9E+09,9E+09,9E+09]];
    CONST robtarget Target_3250:=[[62.178,69.451,0],[0.119542298,0.027125582,0.159127158,0.979618492],[-1,-1,1,0],[9E+09,9E+09,9E+09,9E+09,9E+09,9E+09]];
    CONST robtarget Target_3260:=[[62.756,68.017,0],[0.119542298,0.027125582,0.159127158,0.979618492],[-1,-1,1,0],[9E+09,9E+09,9E+09,9E+09,9E+09,9E+09]];
    CONST robtarget Target_3270:=[[64.884,67.593,0],[0.119542298,0.027125582,0.159127158,0.979618492],[-1,-1,1,0],[9E+09,9E+09,9E+09,9E+09,9E+09,9E+09]];
    CONST robtarget Target_3280:=[[67.801,67.593,0],[0.119542298,0.027125582,0.159127158,0.979618492],[-1,-1,1,0],[9E+09,9E+09,9E+09,9E+09,9E+09,9E+09]];
    CONST robtarget Target_3290:=[[67.801,71.342,0],[0.119542298,0.027125582,0.159127158,0.979618492],[-1,-1,1,0],[9E+09,9E+09,9E+09,9E+09,9E+09,9E+09]];
    CONST robtarget Target_3300:=[[67.801,71.342,-10],[0.119542298,0.027125582,0.159127158,0.979618492],[-1,-1,1,0],[9E+09,9E+09,9E+09,9E+09,9E+09,9E+09]];
    CONST robtarget Target_3310:=[[52.121,75.499,-10],[0.119542298,0.027125582,0.159127158,0.979618492],[-1,-1,1,0],[9E+09,9E+09,9E+09,9E+09,9E+09,9E+09]];
    CONST robtarget Target_3320:=[[52.121,75.499,0],[0.119542298,0.027125582,0.159127158,0.979618492],[-1,-1,1,0],[9E+09,9E+09,9E+09,9E+09,9E+09,9E+09]];
    CONST robtarget Target_3330:=[[46.954,75.499,0],[0.119542298,0.027125582,0.159127158,0.979618492],[-1,-1,1,0],[9E+09,9E+09,9E+09,9E+09,9E+09,9E+09]];
    CONST robtarget Target_3340:=[[46.954,56.819,0],[0.119542298,0.027125582,0.159127158,0.979618492],[-1,-1,1,0],[9E+09,9E+09,9E+09,9E+09,9E+09,9E+09]];
    CONST robtarget Target_3350:=[[52.121,56.819,0],[0.119542298,0.027125582,0.159127158,0.979618492],[-1,-1,1,0],[9E+09,9E+09,9E+09,9E+09,9E+09,9E+09]];
    CONST robtarget Target_3360:=[[52.121,75.499,0],[0.119542298,0.027125582,0.159127158,0.979618492],[-1,-1,1,0],[9E+09,9E+09,9E+09,9E+09,9E+09,9E+09]];
    CONST robtarget Target_3370:=[[52.121,75.499,-10],[0.119542298,0.027125582,0.159127158,0.979618492],[-1,-1,1,0],[9E+09,9E+09,9E+09,9E+09,9E+09,9E+09]];
    CONST robtarget Target_3380:=[[41.672,75.499,-10],[0.119542298,0.027125582,0.159127158,0.979618492],[-1,-1,1,0],[9E+09,9E+09,9E+09,9E+09,9E+09,9E+09]];
    CONST robtarget Target_3390:=[[41.672,75.499,0],[0.119542298,0.027125582,0.159127158,0.979618492],[-1,-1,1,0],[9E+09,9E+09,9E+09,9E+09,9E+09,9E+09]];
    CONST robtarget Target_3400:=[[27.051,75.499,0],[0.119542298,0.027125582,0.159127158,0.979618492],[-1,-1,1,0],[9E+09,9E+09,9E+09,9E+09,9E+09,9E+09]];
    CONST robtarget Target_3410:=[[27.051,72.027,0],[0.119542298,0.027125582,0.159127158,0.979618492],[-1,-1,1,0],[9E+09,9E+09,9E+09,9E+09,9E+09,9E+09]];
    CONST robtarget Target_3420:=[[36.62,72.027,0],[0.119542298,0.027125582,0.159127158,0.979618492],[-1,-1,1,0],[9E+09,9E+09,9E+09,9E+09,9E+09,9E+09]];
    CONST robtarget Target_3430:=[[36.62,68.099,0],[0.119542298,0.027125582,0.159127158,0.979618492],[-1,-1,1,0],[9E+09,9E+09,9E+09,9E+09,9E+09,9E+09]];
    CONST robtarget Target_3440:=[[28.535,68.099,0],[0.119542298,0.027125582,0.159127158,0.979618492],[-1,-1,1,0],[9E+09,9E+09,9E+09,9E+09,9E+09,9E+09]];
    CONST robtarget Target_3450:=[[28.535,64.773,0],[0.119542298,0.027125582,0.159127158,0.979618492],[-1,-1,1,0],[9E+09,9E+09,9E+09,9E+09,9E+09,9E+09]];
    CONST robtarget Target_3460:=[[36.62,64.773,0],[0.119542298,0.027125582,0.159127158,0.979618492],[-1,-1,1,0],[9E+09,9E+09,9E+09,9E+09,9E+09,9E+09]];
    CONST robtarget Target_3470:=[[36.62,60.372,0],[0.119542298,0.027125582,0.159127158,0.979618492],[-1,-1,1,0],[9E+09,9E+09,9E+09,9E+09,9E+09,9E+09]];
    CONST robtarget Target_3480:=[[26.677,60.372,0],[0.119542298,0.027125582,0.159127158,0.979618492],[-1,-1,1,0],[9E+09,9E+09,9E+09,9E+09,9E+09,9E+09]];
    CONST robtarget Target_3490:=[[26.677,56.819,0],[0.119542298,0.027125582,0.159127158,0.979618492],[-1,-1,1,0],[9E+09,9E+09,9E+09,9E+09,9E+09,9E+09]];
    CONST robtarget Target_3500:=[[41.672,56.819,0],[0.119542298,0.027125582,0.159127158,0.979618492],[-1,-1,1,0],[9E+09,9E+09,9E+09,9E+09,9E+09,9E+09]];
    CONST robtarget Target_3510:=[[41.672,75.499,0],[0.119542298,0.027125582,0.159127158,0.979618492],[-1,-1,1,0],[9E+09,9E+09,9E+09,9E+09,9E+09,9E+09]];
    CONST robtarget Target_3520:=[[41.672,75.499,-10],[0.119542298,0.027125582,0.159127158,0.979618492],[-1,-1,1,0],[9E+09,9E+09,9E+09,9E+09,9E+09,9E+09]];
    CONST robtarget Target_3530:=[[22.308,75.499,-10],[0.119542298,0.027125582,0.159127158,0.979618492],[-1,-1,1,0],[9E+09,9E+09,9E+09,9E+09,9E+09,9E+09]];
    CONST robtarget Target_3540:=[[22.308,75.499,0],[0.119542298,0.027125582,0.159127158,0.979618492],[-1,-1,1,0],[9E+09,9E+09,9E+09,9E+09,9E+09,9E+09]];
    CONST robtarget Target_3550:=[[17.255,75.499,0],[0.119542298,0.027125582,0.159127158,0.979618492],[-1,-1,1,0],[9E+09,9E+09,9E+09,9E+09,9E+09,9E+09]];
    CONST robtarget Target_3560:=[[17.255,60.829,0],[0.119542298,0.027125582,0.159127158,0.979618492],[-1,-1,1,0],[9E+09,9E+09,9E+09,9E+09,9E+09,9E+09]];
    CONST robtarget Target_3570:=[[8.518,60.829,0],[0.119542298,0.027125582,0.159127158,0.979618492],[-1,-1,1,0],[9E+09,9E+09,9E+09,9E+09,9E+09,9E+09]];
    CONST robtarget Target_3580:=[[8.518,56.819,0],[0.119542298,0.027125582,0.159127158,0.979618492],[-1,-1,1,0],[9E+09,9E+09,9E+09,9E+09,9E+09,9E+09]];
    CONST robtarget Target_3590:=[[22.308,56.819,0],[0.119542298,0.027125582,0.159127158,0.979618492],[-1,-1,1,0],[9E+09,9E+09,9E+09,9E+09,9E+09,9E+09]];
    CONST robtarget Target_3600:=[[22.308,75.499,0],[0.119542298,0.027125582,0.159127158,0.979618492],[-1,-1,1,0],[9E+09,9E+09,9E+09,9E+09,9E+09,9E+09]];
    CONST robtarget Target_3610:=[[22.308,75.499,-10],[0.119542298,0.027125582,0.159127158,0.979618492],[0,0,0,0],[9E+09,9E+09,9E+09,9E+09,9E+09,9E+09]];
    CONST robtarget Target_3620:=[[94.194,38.558,-10],[0.119542298,0.027125582,0.159127158,0.979618492],[-1,-1,1,0],[9E+09,9E+09,9E+09,9E+09,9E+09,9E+09]];
    CONST robtarget Target_3630:=[[94.194,38.558,0],[0.119542298,0.027125582,0.159127158,0.979618492],[-1,-1,1,0],[9E+09,9E+09,9E+09,9E+09,9E+09,9E+09]];
    CONST robtarget Target_3640:=[[75.235,49.668,0],[0.119542298,0.027125582,0.159127158,0.979618492],[-1,-1,1,0],[9E+09,9E+09,9E+09,9E+09,9E+09,9E+09]];
    CONST robtarget Target_3650:=[[56.071,38.286,0],[0.119542298,0.027125582,0.159127158,0.979618492],[-1,-1,1,0],[9E+09,9E+09,9E+09,9E+09,9E+09,9E+09]];
    CONST robtarget Target_3660:=[[56.071,16.422,0],[0.119542298,0.027125582,0.159127158,0.979618492],[-1,-1,1,0],[9E+09,9E+09,9E+09,9E+09,9E+09,9E+09]];
    CONST robtarget Target_3670:=[[75.083,5.281,0],[0.119542298,0.027125582,0.159127158,0.979618492],[-1,-1,1,0],[9E+09,9E+09,9E+09,9E+09,9E+09,9E+09]];
    CONST robtarget Target_3680:=[[94.194,16.631,0],[0.119542298,0.027125582,0.159127158,0.979618492],[-1,-1,1,0],[9E+09,9E+09,9E+09,9E+09,9E+09,9E+09]];
    CONST robtarget Target_3690:=[[94.194,38.558,0],[0.119542298,0.027125582,0.159127158,0.979618492],[-1,-1,1,0],[9E+09,9E+09,9E+09,9E+09,9E+09,9E+09]];
    CONST robtarget Target_3930:=[[67.472477576,40.059752487,-14.996049097],[0.119542298,0.027125582,0.159127158,0.979618492],[-2,-1,1,0],[9E+09,9E+09,9E+09,9E+09,9E+09,9E+09]];
    CONST robtarget Target_3700:=[[94.194,38.558,-10],[0.119542298,0.027125582,0.159127158,0.979618492],[-1,-1,1,0],[9E+09,9E+09,9E+09,9E+09,9E+09,9E+09]];
    CONST robtarget Target_3710:=[[89.358,36.21,-10],[0.119542298,0.027125582,0.159127158,0.979618492],[-1,-1,1,0],[9E+09,9E+09,9E+09,9E+09,9E+09,9E+09]];
    CONST robtarget Target_3720:=[[89.358,36.21,0],[0.119542298,0.027125582,0.159127158,0.979618492],[-1,-1,1,0],[9E+09,9E+09,9E+09,9E+09,9E+09,9E+09]];
    CONST robtarget Target_3730:=[[75.235,44.113,0],[0.119542298,0.027125582,0.159127158,0.979618492],[-1,-1,1,0],[9E+09,9E+09,9E+09,9E+09,9E+09,9E+09]];
    CONST robtarget Target_3740:=[[72.307,41.696,0],[0.119542298,0.027125582,0.159127158,0.979618492],[-1,-1,1,0],[9E+09,9E+09,9E+09,9E+09,9E+09,9E+09]];
    CONST robtarget Target_3750:=[[70.636,38.286,0],[0.119542298,0.027125582,0.159127158,0.979618492],[-1,-1,1,0],[9E+09,9E+09,9E+09,9E+09,9E+09,9E+09]];
    CONST robtarget Target_3760:=[[81.246,14.208,0],[0.119542298,0.027125582,0.159127158,0.979618492],[-1,-1,1,0],[9E+09,9E+09,9E+09,9E+09,9E+09,9E+09]];
    CONST robtarget Target_3770:=[[85.302,16.617,0],[0.119542298,0.027125582,0.159127158,0.979618492],[-1,-1,1,0],[9E+09,9E+09,9E+09,9E+09,9E+09,9E+09]];
    CONST robtarget Target_3780:=[[89.358,19.026,0],[0.119542298,0.027125582,0.159127158,0.979618492],[-1,-1,1,0],[9E+09,9E+09,9E+09,9E+09,9E+09,9E+09]];
    CONST robtarget Target_3790:=[[89.358,36.21,0],[0.119542298,0.027125582,0.159127158,0.979618492],[-1,-1,1,0],[9E+09,9E+09,9E+09,9E+09,9E+09,9E+09]];
    CONST robtarget Target_3800:=[[89.358,36.21,-10],[0.119542298,0.027125582,0.159127158,0.979618492],[-1,-1,1,0],[9E+09,9E+09,9E+09,9E+09,9E+09,9E+09]];
    CONST robtarget Target_3810:=[[68.77,34.464,-10],[0.119542298,0.027125582,0.159127158,0.979618492],[-1,-1,1,0],[9E+09,9E+09,9E+09,9E+09,9E+09,9E+09]];
    CONST robtarget Target_3820:=[[68.77,34.464,0],[0.119542298,0.027125582,0.159127158,0.979618492],[-1,-1,1,0],[9E+09,9E+09,9E+09,9E+09,9E+09,9E+09]];
    CONST robtarget Target_3830:=[[62.422,17.88,0],[0.119542298,0.027125582,0.159127158,0.979618492],[-1,-1,1,0],[9E+09,9E+09,9E+09,9E+09,9E+09,9E+09]];
    CONST robtarget Target_3840:=[[74.993,10.536,0],[0.119542298,0.027125582,0.159127158,0.979618492],[-1,-1,1,0],[9E+09,9E+09,9E+09,9E+09,9E+09,9E+09]];
    CONST robtarget Target_3850:=[[77.735,12.123,0],[0.119542298,0.027125582,0.159127158,0.979618492],[-1,-1,1,0],[9E+09,9E+09,9E+09,9E+09,9E+09,9E+09]];
    CONST robtarget Target_3860:=[[68.77,34.464,0],[0.119542298,0.027125582,0.159127158,0.979618492],[-1,-1,1,0],[9E+09,9E+09,9E+09,9E+09,9E+09,9E+09]];
    CONST robtarget Target_3870:=[[68.77,34.464,-10],[0.119542298,0.027125582,0.159127158,0.979618492],[-1,-1,1,0],[9E+09,9E+09,9E+09,9E+09,9E+09,9E+09]];
    CONST robtarget Target_3880:=[[67.293,40.162,-10],[0.119542298,0.027125582,0.159127158,0.979618492],[-1,-1,1,0],[9E+09,9E+09,9E+09,9E+09,9E+09,9E+09]];
    CONST robtarget Target_3890:=[[67.293,40.162,0],[0.119542298,0.027125582,0.159127158,0.979618492],[-1,-1,1,0],[9E+09,9E+09,9E+09,9E+09,9E+09,9E+09]];
    CONST robtarget Target_3900:=[[60.509,36.21,0],[0.119542298,0.027125582,0.159127158,0.979618492],[-1,-1,1,0],[9E+09,9E+09,9E+09,9E+09,9E+09,9E+09]];
    CONST robtarget Target_3910:=[[60.509,24.537,0],[0.119542298,0.027125582,0.159127158,0.979618492],[-1,-1,1,0],[9E+09,9E+09,9E+09,9E+09,9E+09,9E+09]];
    CONST robtarget Target_3920:=[[67.293,40.162,0],[0.119542298,0.027125582,0.159127158,0.979618492],[-1,-1,1,0],[9E+09,9E+09,9E+09,9E+09,9E+09,9E+09]];
    PERS tooldata Marcador:=[TRUE,[[0,-100.213,125.309],[0.165634,0.0951553,-0.490794,0.850078]],[1,[0,0,1],[1,0,0,0],0,0,0]];
    TASK PERS wobjdata Pastel:=[FALSE,TRUE,"",[[0,0,0],[1,0,0,0]],[[-69.127,-648.568,653.794],[0.0103063,-0.999781,-0.00319575,-0.0179544]]];
    TASK PERS wobjdata WNaranja:=[FALSE,TRUE,"",[[0,0,0],[1,0,0,0]],[[-69.1267,-648.568,653.794],[0.0103056,-0.999781,-0.00319482,-0.0179566]]];
    !CONST robtarget HOME:=[[685.456722929,-542.846554009,72.789258876],[0.784186308,-0.518748937,0.327912498,0.091786542],[-1,0,-1,0],[9E+09,9E+09,9E+09,9E+09,9E+09,9E+09]];

    CONST robtarget HOME:=[[685.456722929,-542.846554009,72.789258876],[0.784186308,-0.518748937,0.327912498,0.091786542],[-1,-1,1,0],[9E+09,9E+09,9E+09,9E+09,9E+09,9E+09]];
    CONST robtarget Aproximacion:=[[140.364595003,1.820278874,-22.05975894],[0.119542298,0.027125582,0.159127158,0.979618492],[-1,-1,1,0],[9E+09,9E+09,9E+09,9E+09,9E+09,9E+09]];
    CONST robtarget Target_3940:=[[68.00538685,-48.442633556,-13.16160056],[0.119542298,0.027125582,0.159127158,0.979618492],[-2,-1,1,0],[9E+09,9E+09,9E+09,9E+09,9E+09,9E+09]];

    CONST jointtarget HOME0:=[[0,0,0,0,0,0],[9E+09,9E+09,9E+09,9E+09,9E+09,9E+09]];
    CONST jointtarget SINGBREAK:=[[0,0,0,0,30,0],[9E+09,9E+09,9E+09,9E+09,9E+09,9E+09]];

